Staubli VAL3: _getP2PDistance.pgx

public program _getP2PDistance(point x_pPoint, point x_pHere, num& x_nP2PDsts[])
  local num l_nResult[14]
begin
  x_nP2PDsts=distance(position(x_pPoint,world),position(x_pHere,world))

end
